// TIA Portal V15.1 export
// export: Created 2020-12-09T10:31:54.8859095Z, ExportSetting WithDefaults, WithReadOnly, DisplayName Totally Integrated Automation Portal, DisplayVersion V15.1 Update 4, DisplayName TIA Portal Openness, DisplayVersion V15.1, DisplayName SINAMICS Startdrive Advanced, DisplayVersion V15.1 Update3, DisplayName SINAMICS Startdrive G110M, G120, G120C, G120D, G120P, DisplayVersion V15.1 Update3, DisplayName SINAMICS Startdrive G130, G150, S120, S150, SINAMICS MV, S210, DisplayVersion V15.1 Update3, DisplayName STEP 7 Professional, DisplayVersion V15.1 Update 4, DisplayName STEP 7 Safety, DisplayVersion V15.1, DisplayName WinCC Professional, DisplayVersion V15.1 Update 4
FUNCTION "PROAUTOMATOR_EV" : Void   // FC7, LAD
{ S7_Optimized_Access := 'TRUE' }
VERSION : 0.1
// stored: AutoNumber true, CodeModifiedDate 2020-12-09T10:31:10.2667692Z, CompileDate 2020-12-09T10:31:25.5011439Z, CreationDate 2020-12-09T10:30:25.6105189Z, HandleErrorsWithinBlock false, InterfaceModifiedDate 2020-12-09T10:30:25.6105189Z, IsConsistent true, IsIECCheckEnabled false, IsKnowHowProtected false, IsWriteProtected false, LibraryConformanceStatus Warning: The object contains access to global data blocks., ModifiedDate 2020-12-09T10:31:10.2667692Z, ParameterModified 2020-12-09T10:30:25.6105189Z, PLCSimAdvancedSupport true, SetENOAutomatically False, StructureModified 2020-12-09T10:30:25.6105189Z, UDAEnableTagReadback false
BEGIN

REGION Network 1: {AUTOGENERATED BEGIN} - DO NOT REMOVE COMMENT
END_REGION

REGION Network 2: {AUTOGENERATED END} - DO NOT REMOVE COMMENT
END_REGION

REGION Network 3: Stazione in manuale
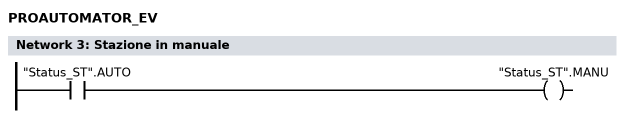
   RUNG wire#powerrail
      Contact( "Status_ST".AUTO )
      Coil( "Status_ST".MANU )
   END_RUNG
   // the same network as SCL:
   "Status_ST".MANU := "Status_ST".AUTO;
END_REGION
END_FUNCTION
